// Reads a bytes field value from the input.
FUNCTION F_ReadBytes : HRESULT
VAR_INPUT CONSTANT
    aBuffer : ARRAY [*] OF BYTE;   
END_VAR
VAR_IN_OUT
    stState : ST_ParserInternalState;
    aBytes  : ARRAY[*] OF BYTE;
END_VAR
VAR
    nLength : UDINT;
END_VAR

F_ReadBytes := S_OK;

F_ReadBytes := F_ParseLength(aBuffer, stState, nLength=> nLength);
IF FAILED(F_ReadBytes) THEN
    RETURN;
END_IF

F_ReadBytes := F_ReadRawBytes(aBuffer, nLength, stState, aBytes);

END_FUNCTION

(* stored: Version 1.1.0.1
   POU F_ReadBytes: Id {fe8d4fa5-1dc0-4cb1-bc5f-aa95aabb97fd}, SpecialFunc None *)
